// TIA Portal V17 export
// export: Created 2026-04-13T11:12:44.3447416Z, ExportSetting WithDefaults, DisplayName Totally Integrated Automation Portal, DisplayVersion V17 Update 4, DisplayName TIA Portal Openness, DisplayVersion V17 Update 4, DisplayName TIA Portal Version Control Interface, DisplayVersion V17, DisplayName SINAMICS Startdrive Advanced, DisplayVersion V17, DisplayName SINAMICS Startdrive G130, G150, S120, S150, SINAMICS MV, S210, DisplayVersion V17, DisplayName SINAMICS Startdrive G110M, G120, G120C, G120D, G120P, G115D, DisplayVersion V17, DisplayName STEP 7 Professional, DisplayVersion V17 Update 4, DisplayName STEP 7 Safety, DisplayVersion V17, DisplayName WinCC Professional, DisplayVersion V17 Update 4
DATA_BLOCK "A3-电机控制_DB"   // DB5
VERSION : 0.1
// stored: AutoNumber true, DBAccessibleFromOPCUA true, DBAccessibleFromWebserver true, InstanceOfName A3-电机控制, InstanceOfType FB
"A3-电机控制"
   // VAR
   //    进料泵控制 { S7_SetPoint := 'True'} : "A4-蠕动泵控制";
   //    引风频率 { S7_SetPoint := 'True'} : "A4--电机控制";
   //    送风频率 { S7_SetPoint := 'True'} : "A4--电机控制";
   //    离心雾化 { S7_SetPoint := 'True'} : "A4--电机控制";
   // END_VAR
BEGIN
END_DATA_BLOCK
